// Struckig
// Copyright (C) 2022 Stefan Besler

// This program is free software: you can redistribute it and/or modify
// it under the terms of the GNU General Public License as published by
// the Free Software Foundation, either version 3 of the License, or
// (at your option) any later version.

// This program is distributed in the hope that it will be useful,
// but WITHOUT ANY WARRANTY; without even the implied warranty of
// MERCHANTABILITY or FITNESS FOR A PARTICULAR PURPOSE.  See the
// GNU General Public License for more details.
//
// You should have received a copy of the GNU General Public License
// along with THIS PROGRAM.  IF NOT, see <http://www.gnu.org/licenses/>.
{attribute 'hide'}
/// Internal bubble-sort helper for `LREAL` arrays.
/// Returns sorted index positions in `indicesSorted` without modifying input `data`.
FUNCTION BubbleSortLreal : BOOL
VAR_INPUT
  data : POINTER TO LREAL; //< Input unsorted array.
  size : INT; //< Number of elements in `data`.
  indicesSorted : POINTER TO INT; //< Output sorted indices.
END_VAR
VAR
  i, j, h : INT;
END_VAR

FOR i:=0 TO size
DO
  indicesSorted[i] := i;
END_FOR

// Bubblesort possible_t_syncs from best to worst
FOR i:=0 TO size-1
DO
  FOR j:=0 TO size-1-i
  DO  
    IF data[indicesSorted[j]] > data[indicesSorted[j+1]]
    THEN
      h := indicesSorted[j];
      indicesSorted[j] := indicesSorted[j+1];
      indicesSorted[j+1] := h;     
		END_IF
  END_FOR
END_FOR

END_FUNCTION

(* stored: Version 1.1.0.1
   POU BubbleSortLreal: Id {019830ac-0aa6-4391-9a8a-478037ed79fe}, SpecialFunc None *)
